Staubli VAL3: clkValve13.pgx

program clkValve13()
begin
  call toggleValve(13)
end
